// TIA Portal V17 export
// export: Created 2023-04-07T09:30:35.1801872Z, ExportSetting WithDefaults, DisplayName Totally Integrated Automation Portal, DisplayVersion V17 Update 4, DisplayName TIA Portal Openness, DisplayVersion V17 Update 4, DisplayName TIA Portal Version Control Interface, DisplayVersion V17, DisplayName STEP 7 Professional, DisplayVersion V17 Update 4, DisplayName STEP 7 Safety, DisplayVersion V17, DisplayName WinCC Professional, DisplayVersion V17 Update 4
TYPE "R_PE"
// stored: IsFailsafeCompliant false
   STRUCT
      diCurrentFault : UInt := 0;   // Register 41001 / 41001
      diCurrentFaultModule : UInt := 0;   // Register 41002 / 41002
      diCurrentWarning : UInt := 0;   // Register 41003 / 41003
      iCurrentStatus : Int := 0;   // Register 41004 / 41004
      xStartCodnition_all : Bool := false;   // Register 40928
      xStartCodnition_V : Bool := false;   // Register 40929
      xStartCondition_f : Bool := false;   // Register 41041 / 41005
      xStartCondition_Vdc : Bool := false;   // Register 41042 / 41006
      xStartCondition_MVcell : Bool := false;   // Register 41043 / 41007
      xStartCondition_P : Bool := false;   // Register 41044 / 41008
      iAcSwitchStatus : Int := 0;   // Register 40632 / 41009
      iMVswitchStatus : Int := 0;   // Register 40634 / 41010
      iMVgenswitchStatus : Int := 0;   // Register 40636 / 41011
      iMVearthswitchStatus : Int := 0;   // Register 40637 / 41013
      iDC1switchStatus : Int := 0;   // Register 40638 / 41014
      iDC2switchStatus : Int := 0;   // Register 40639 / 41015
      iDC3switchStatus : Int := 0;   // Register 40640 / 41021
      iDC4switchStatus : Int := 0;   // Register 40641 / 41026
      bStatusDspRJ13 : Byte := 0;   // Register 41084 / 41027
      bStatusDspRJ14 : Byte := 0;   // Register 41085 / 41028
      bStatusDspRJ15 : Byte := 0;   // Register 41086
      bStatusDspRJ16 : Byte := 0;   // Register 41087
      bStatusDspRJ20 : Byte := 0;   // Register 41090
      iMV_PT100_1 : Int := 0;   // Register 41109
      iMV_PT100_2 : Int := 0;   // Register 41110
      iMV_PT100_3 : Int := 0;   // Register 41111
      iP_control : Int := 0;   // Register 41113
      iQ_control : Int := 0;   // Register 41114
      iInputPower_1 : Int := 0;   // Register 41373 / 41029
      iInputPower_2 : Int := 0;   // Register 41374 / 41030
      iInputPower_3 : Int := 0;   // Register 41375 / 41031
      iInputPower_4 : Int := 0;   // 41032 / Register 41376
      rI_DC1 : Real := 0.0;   // 41033 / Register 41377
      rI_DC2 : Real := 0.0;   // 41034 / Register 41378
      rI_DC3 : Real := 0.0;   // 41036 / Register 41379
      rI_DC4 : Real := 0.0;   // 41037 / Register 41380
      rDCvoltageBus_1 : Real := 0.0;   // 41039 / Register 41381
      rDCvoltageBus_2 : Real := 0.0;   // 41040 / Register 41382
      rDCvoltageBus_3 : Real := 0.0;   // Register 41383 / 41141
      rDCvoltageBus_4 : Real := 0.0;   // Register 41384 / 41142
      rDCvoltageExt_1 : Real := 0.0;   // Register 41385 / 41251
      rDCvoltageExt_2 : Real := 0.0;   // Register 41386 / 47402
      rDCvoltageExt_3 : Real := 0.0;   // Register 41387 / 47402
      rDCvoltageExt_4 : Real := 0.0;   // Register 41388 / 47410
      rDCvoltageLast_1 : Real := 0.0;   // Register 41389 / 47411
      rDCvoltageLast_2 : Real := 0.0;   // Register 41390 / 47416
      rDCvoltageLast_3 : Real := 0.0;   // Register 41391
      rDCvoltageLast_4 : Real := 0.0;   // Register 41392
      rMVgridVoltage_RS : Real := 0.0;   // Register 44301
      rMVgridVoltage_ST : Real := 0.0;   // Register 44302
      rMVgridVoltage_TR : Real := 0.0;   // Register 44303 / 41015
      rMVgridCurrent_I1 : Real := 0.0;   // Register 44304
      rMVgridCurrent_I2 : Real := 0.0;   // Register 44305
      rMVgridCurrent_I3 : Real := 0.0;   // Register 44306
      iMV_P : Int := 0;   // Register 44307
      iMV_Q : Int := 0;   // Register 44308
      uiMV_S : UInt := 0;   // Register 44309
      rMVcosphi : Real := 0.0;   // Register 44310
      rLVgridVoltage_RS : Real := 0.0;   // Register 44321
      rLVgridVoltage_ST : Real := 0.0;   // Register 44322
      rLVgridVoltage_TR : Real := 0.0;   // Register 44323
      rLVgridCurrent_I1 : Real := 0.0;   // Register 44324
      rLVgridCurrent_I2 : Real := 0.0;   // Register 44325
      rLVgridCurrent_I3 : Real := 0.0;   // Register 44326
      iLV_P : Int := 0;   // Register 44327
      iLV_Q : Int := 0;   // Register 44328
      uiLV_S : UInt := 0;   // Register 44329
      rLVcosphi : Real := 0.0;   // Register 44330
      xGridSequency : Bool;   // Register 44331
      rGridFreq : Real := 0.0;   // Register 44332
      wRunningModules : Word;   // Register 46501
      bNumRunningModules : Byte;   // Register 46502
      bNextStartModule : Byte;   // Register 46503
      wModuleStartStop : Word;   // Register 46504
      wModulesEnableReg : Word;   // Register 46505
      Module_1 { S7_SetPoint := 'True'} : "MODULE_PE";
      Module_2 { S7_SetPoint := 'True'} : "MODULE_PE";
      Module_3 { S7_SetPoint := 'True'} : "MODULE_PE";
      Module_4 { S7_SetPoint := 'True'} : "MODULE_PE";
   END_STRUCT;
END_TYPE
